(*
SPDX-FileCopyrightText: Â© 2026 Oleksandr Tiutyk <trofimich@gmail.com>
SPDX-License-Identifier: MIT
License: https://opensource.org/license/mit
*)

(*!
<summary>Read-only contract for a digital input automation component.</summary>
<description>
Provides access to logical boolean state, change detection and electrical contact configuration.
</description>
*)

INTERFACE IReadOnlyDigitalInput EXTENDS TOF_Automation.IInputLeafAutomationComponent

(*!
<summary>Indicates whether the logical Value has changed compared to the previous cycle.</summary>
*)
{attribute 'monitoring' := 'call'}
PROPERTY Changed : BOOL
GET
END_GET
END_PROPERTY

(*!
<summary>Gets electrical contact configuration (normally open or normally closed).</summary>
*)
{attribute 'monitoring' := 'call'}
PROPERTY ContactType : CONTACT_TYPE
GET
END_GET
END_PROPERTY

(*!
<summary>Gets current evaluated logical state of the input signal.</summary>
*)
{attribute 'monitoring' := 'call'}
PROPERTY Value : BOOL
GET
END_GET
END_PROPERTY

END_INTERFACE

(* stored: Version 1.1.0.1
   Itf IReadOnlyDigitalInput: Id {0e003d9a-9e50-45cd-ba08-9b230647b62a}
   Property Changed: Id {9dfeebaf-2fa2-4766-acbd-c5332314353f}
   Get Get: Id {1a7feeca-815a-46d7-b785-0b71640f7501}
   Property ContactType: Id {26bb28e2-69d5-41c5-a4e9-55529b93ddba}
   Get Get: Id {901186a8-8bc5-40a3-8257-70bf2029c8d0}
   Property Value: Id {76a6088e-f0a2-4288-be31-c3df6ee448b5}
   Get Get: Id {d3195ff5-7740-4efc-9751-6036d3c2571f} *)
